// TIA Portal V20 export
VAR_GLOBAL   // PLC tag table "AXIS tags"
   Brugaansturing_axis_IN AT %I256.0 : "PD_TEL3_IN";
   Brugaansturing_axis_OUT AT %Q256.0 : "PD_TEL3_OUT";
END_VAR
